// TIA Portal V20 export
FUNCTION_BLOCK "FB_DigitalOutputsSonplas"   // FB213, SCL
{ S7_Optimized_Access := 'TRUE' }
// stored: AutoNumber false, MemoryReserve 100, SetENOAutomatically false
   VAR
      Free_Q0_0 : "FB_DigitalOutput";
      Operating_Counter : "FB_DigitalOutput";
      General_Air_Valve : "FB_DigitalOutput";
      Smart_Line_Disable : "FB_DigitalOutput";
      Machine_Light : "FB_DigitalOutput";
      Machine_Light_Back : "FB_DigitalOutput";
      Light_Tower_Orange : "FB_DigitalOutput";
      Light_Tower_Red : "FB_DigitalOutput";
      Light_Tower_Blue : "FB_DigitalOutput";
      Light_Tower_Green : "FB_DigitalOutput";
      Light_Tower_White : "FB_DigitalOutput";
      Backlight : "FB_DigitalOutput";
      Free_Q1_4 : "FB_DigitalOutput";
      Infeed_ON : "FB_DigitalOutput";
      Axis_Activation : "FB_DigitalOutput";
      Buzzer_Activation : "FB_DigitalOutput";
      Elbaron_Power_ON : "FB_DigitalOutput";
      Observation_Camera_Light : "FB_DigitalOutput";
      Laser_External_Door_Opening : "FB_DigitalOutput";
      Cooling_Start : "FB_DigitalOutput";
      X_Axis_Brake_Activation : "FB_DigitalOutput";
      Y_Axis_Brake_Activation : "FB_DigitalOutput";
      Axis_B_TeachIn_Clamping_Part : "FB_DigitalOutput";
      EPO_UPS : "FB_DigitalOutput";
      Head_Laser_Start : "FB_DigitalOutput";
      Head_Laser_Stop : "FB_DigitalOutput";
      Axis_2_Power_Contactor : "FB_DigitalOutput";
      GasAssistOn : "FB_DigitalOutput";
      Smart_Line_Reset : "FB_DigitalOutput";
      XY_Axis_Power_Contactor : "FB_DigitalOutput";
      Laser_Air_Pressure_Process : "FB_DigitalOutput";
      Bus60V_Power_Contactor : "FB_DigitalOutput";
      Free_Q4_0 : "FB_DigitalOutput";
      Free_Q4_1 : "FB_DigitalOutput";
      Free_Q4_2 : "FB_DigitalOutput";
      Free_Q4_3 : "FB_DigitalOutput";
      Load_Clamp_Closing : "FB_DigitalOutput";
      Load_Clamp_Opening : "FB_DigitalOutput";
      Unload_Clamp_Closing : "FB_DigitalOutput";
      Unload_Clamp_Opening : "FB_DigitalOutput";
      Clamping_Opening : "FB_DigitalOutput";
      Clamping_Closing : "FB_DigitalOutput";
      B_Axis_Brake_Release : "FB_DigitalOutput";
      Suction : "FB_DigitalOutput";
      Free_Q5_4 : "FB_DigitalOutput";
      Free_Q5_5 : "FB_DigitalOutput";
      Free_Q5_6 : "FB_DigitalOutput";
      Free_Q5_7 : "FB_DigitalOutput";
      External_Gate_Closing : "FB_DigitalOutput";
      External_Gate_Opening : "FB_DigitalOutput";
      Internal_Gate_Closing : "FB_DigitalOutput";
      Internal_Gate_Opening : "FB_DigitalOutput";
      PowerMeter_Retract : "FB_DigitalOutput";
      PowerMeter_Advance : "FB_DigitalOutput";
      Blowing : "FB_DigitalOutput";
      Free_Q8_7 : "FB_DigitalOutput";
      Free_Q9_0 : "FB_DigitalOutput";
      Free_Q9_1 : "FB_DigitalOutput";
      Free_Q9_2 : "FB_DigitalOutput";
      Free_Q9_3 : "FB_DigitalOutput";
      Free_Q9_4 : "FB_DigitalOutput";
      Free_Q9_5 : "FB_DigitalOutput";
      Free_Q9_6 : "FB_DigitalOutput";
      Free_Q9_7 : "FB_DigitalOutput";
      Sonplas_DiagDPCoupler { S7_SetPoint := 'True'} : "FB_DigitalOutput";
      Sonplas_Ready { S7_SetPoint := 'True'} : "FB_DigitalOutput";
      Sonplas_NoEStop { S7_SetPoint := 'True'} : "FB_DigitalOutput";
      Sonplas_DoorsClosed { S7_SetPoint := 'True'} : "FB_DigitalOutput";
      Sonplas_RunError { S7_SetPoint := 'True'} : "FB_DigitalOutput";
      Sonplas_Free_Q200_5 { S7_SetPoint := 'True'} : "FB_DigitalOutput";
      Sonplas_Free_Q200_6 { S7_SetPoint := 'True'} : "FB_DigitalOutput";
      Sonplas_Free_Q200_7 { S7_SetPoint := 'True'} : "FB_DigitalOutput";
      Sonplas_Free_Q201_0 { S7_SetPoint := 'True'} : "FB_DigitalOutput";
      Sonplas_Free_Q201_1 { S7_SetPoint := 'True'} : "FB_DigitalOutput";
      Sonplas_Free_Q201_2 { S7_SetPoint := 'True'} : "FB_DigitalOutput";
      Sonplas_Free_Q201_3 { S7_SetPoint := 'True'} : "FB_DigitalOutput";
      Sonplas_Free_Q201_4 { S7_SetPoint := 'True'} : "FB_DigitalOutput";
      Sonplas_Free_Q201_5 { S7_SetPoint := 'True'} : "FB_DigitalOutput";
      Sonplas_Free_Q201_6 { S7_SetPoint := 'True'} : "FB_DigitalOutput";
      Sonplas_Free_Q201_7 { S7_SetPoint := 'True'} : "FB_DigitalOutput";
      Sonplas_Shuttle1InPos { S7_SetPoint := 'True'} : "FB_DigitalOutput";
      Sonplas_Free_Q202_1 { S7_SetPoint := 'True'} : "FB_DigitalOutput";
      Sonplas_Free_Q202_2 { S7_SetPoint := 'True'} : "FB_DigitalOutput";
      Sonplas_Free_Q202_3 { S7_SetPoint := 'True'} : "FB_DigitalOutput";
      Sonplas_Free_Q202_4 { S7_SetPoint := 'True'} : "FB_DigitalOutput";
      Sonplas_Free_Q202_5 { S7_SetPoint := 'True'} : "FB_DigitalOutput";
      Sonplas_Part1OK { S7_SetPoint := 'True'} : "FB_DigitalOutput";
      Sonplas_Part1NOK { S7_SetPoint := 'True'} : "FB_DigitalOutput";
      Sonplas_Shuttle2InPos { S7_SetPoint := 'True'} : "FB_DigitalOutput";
      Sonplas_Free_Q203_1 { S7_SetPoint := 'True'} : "FB_DigitalOutput";
      Sonplas_Free_Q203_2 { S7_SetPoint := 'True'} : "FB_DigitalOutput";
      Sonplas_Free_Q203_3 { S7_SetPoint := 'True'} : "FB_DigitalOutput";
      Sonplas_Free_Q203_4 { S7_SetPoint := 'True'} : "FB_DigitalOutput";
      Sonplas_Free_Q203_5 { S7_SetPoint := 'True'} : "FB_DigitalOutput";
      Sonplas_Part2OK { S7_SetPoint := 'True'} : "FB_DigitalOutput";
      Sonplas_Part2NOK { S7_SetPoint := 'True'} : "FB_DigitalOutput";
      Sonplas_ResultAccepted { S7_SetPoint := 'True'} : "FB_DigitalOutput";
      Sonplas_Free_Q244_1 { S7_SetPoint := 'True'} : "FB_DigitalOutput";
      Sonplas_Free_Q244_2 { S7_SetPoint := 'True'} : "FB_DigitalOutput";
      Sonplas_Free_Q244_3 { S7_SetPoint := 'True'} : "FB_DigitalOutput";
      Sonplas_Free_Q244_4 { S7_SetPoint := 'True'} : "FB_DigitalOutput";
      Sonplas_Free_Q244_5 { S7_SetPoint := 'True'} : "FB_DigitalOutput";
      Sonplas_Free_Q244_6 { S7_SetPoint := 'True'} : "FB_DigitalOutput";
      Sonplas_Free_Q244_7 { S7_SetPoint := 'True'} : "FB_DigitalOutput";
   END_VAR
BEGIN
   REGION Description head
       //==================================================================================
       // POSALUX Swiss SA / (C) Copyright 2025
       //----------------------------------------------------------------------------------
       // Title: Digital Ouputs mapping
       // Comment/Function: Sonplas Digital Ouputs mapping
       // Author: Fabien WALDT
       // Engineering: TIA Portal v17
       //----------------------------------------------------------------------------------
       // Change log table:
       // Version  | Date     | Expert in charge | Changes applied
       //----------------------------------------------------------------------------------
       // 00.00.01 | 20250423 | WFA              | First released version
       //==================================================================================
   END_REGION

   REGION Operating modes AND parts exchange
       #Sonplas_DiagDPCoupler(oHWStatus => "DQ_SonplasDiagDPCoupler");
       #Sonplas_Ready(oHWStatus => "DQ_SonplasReady");
       #Sonplas_NoEStop(oHWStatus => "DQ_SonplasNoEStop");
       #Sonplas_DoorsClosed(oHWStatus => "DQ_SonplasDoorsClosed");
       #Sonplas_RunError(oHWStatus => "DQ_SonplasRunError");
       #Sonplas_Free_Q200_5(oHWStatus => "DQ_SonplasFreeQ200_5");
       #Sonplas_Free_Q200_6(oHWStatus => "DQ_SonplasFreeQ200_6");
       #Sonplas_Free_Q200_7(oHWStatus => "DQ_SonplasFreeQ200_7");
       // 
       #Sonplas_Free_Q201_0(oHWStatus => "DQ_SonplasFreeQ201_0");
       #Sonplas_Free_Q201_1(oHWStatus => "DQ_SonplasFreeQ201_1");
       #Sonplas_Free_Q201_2(oHWStatus => "DQ_SonplasFreeQ201_2");
       #Sonplas_Free_Q201_3(oHWStatus => "DQ_SonplasFreeQ201_3");
       #Sonplas_Free_Q201_4(oHWStatus => "DQ_SonplasFreeQ201_4");
       #Sonplas_Free_Q201_5(oHWStatus => "DQ_SonplasFreeQ201_5");
       #Sonplas_Free_Q201_6(oHWStatus => "DQ_SonplasFreeQ201_6");
       #Sonplas_Free_Q201_7(oHWStatus => "DQ_SonplasFreeQ201_7");
   END_REGION

   REGION Part exchange
       #Sonplas_Shuttle1InPos(oHWStatus => "DQ_SonplasShuttle1InPos");
       #Sonplas_Free_Q202_1(oHWStatus => "DQ_SonplasFreeQ202_1");
       #Sonplas_Free_Q202_2(oHWStatus => "DQ_SonplasFreeQ202_2");
       #Sonplas_Free_Q202_3(oHWStatus => "DQ_SonplasFreeQ202_3");
       #Sonplas_Free_Q202_4(oHWStatus => "DQ_SonplasFreeQ202_4");
       #Sonplas_Free_Q202_5(oHWStatus => "DQ_SonplasFreeQ202_5");
       #Sonplas_Part1OK(oHWStatus => "DQ_SonplasPart1OK");
       #Sonplas_Part1NOK(oHWStatus => "DQ_SonplasPart1NOK");
       // 
       #Sonplas_Shuttle2InPos(oHWStatus => "DQ_SonplasShuttle2InPos");
       #Sonplas_Free_Q203_1(oHWStatus => "DQ_SonplasFreeQ203_1");
       #Sonplas_Free_Q203_2(oHWStatus => "DQ_SonplasFreeQ203_2");
       #Sonplas_Free_Q203_3(oHWStatus => "DQ_SonplasFreeQ203_3");
       #Sonplas_Free_Q203_4(oHWStatus => "DQ_SonplasFreeQ203_4");
       #Sonplas_Free_Q203_5(oHWStatus => "DQ_SonplasFreeQ203_5");
       #Sonplas_Part2OK(oHWStatus => "DQ_SonplasPart2OK");
       #Sonplas_Part2NOK(oHWStatus => "DQ_SonplasPart2NOK");
   END_REGION

   REGION Measure
       #Sonplas_ResultAccepted(oHWStatus => "DQ_SonplasResultAccepted");
       #Sonplas_Free_Q244_1(oHWStatus => "DQ_SonplasFreeQ244_1");
       #Sonplas_Free_Q244_2(oHWStatus => "DQ_SonplasFreeQ244_2");
       #Sonplas_Free_Q244_3(oHWStatus => "DQ_SonplasFreeQ244_3");
       #Sonplas_Free_Q244_4(oHWStatus => "DQ_SonplasFreeQ244_4");
       #Sonplas_Free_Q244_5(oHWStatus => "DQ_SonplasFreeQ244_5");
       #Sonplas_Free_Q244_6(oHWStatus => "DQ_SonplasFreeQ244_6");
       #Sonplas_Free_Q244_7(oHWStatus => "DQ_SonplasFreeQ244_7");
   END_REGION
END_FUNCTION_BLOCK
